VISUALIZATION SingleFixture  // 1120x220
END_VISUALIZATION

(* stored: Version 1.1.0.1, ProductVersion 3.1.4024.9
   Visu SingleFixture: Id {1fd19add-5656-4611-aaf5-22c8f29453bd} *)
